// TIA Portal V21 export
FUNCTION "Cabinet_Management" : Void   // FC1, LAD
{ S7_Optimized_Access := 'TRUE' }
// stored: SetENOAutomatically false
   VAR_TEMP
      Phase_monitor_OK : Bool;
      Auxiliary_sevices_OK : Bool;
      "400V_protections_OK" : Bool;
      "400V_power_lines_activated" : Bool;
      Aux_emergencies : Bool;
      Emergencies_OK : Bool;
      Aux_cabinet_OK : Bool;
      Cabinet_OK : Bool;
      Heater_OK : Bool;
      Insulation_Monitor_OK : Bool;
      Power_wrapping_machine_OK : Bool;
      Power_fast_doors_OK : Bool;
      Facility_fault : Bool;
      Summary_fault : Bool;
   END_VAR
   VAR_TEMP   // added for the SCL form of the ladder/FBD networks
      _w1 : Bool;
      _w2 : Bool;
   END_VAR
BEGIN

REGION Network 1: Cabinet power control
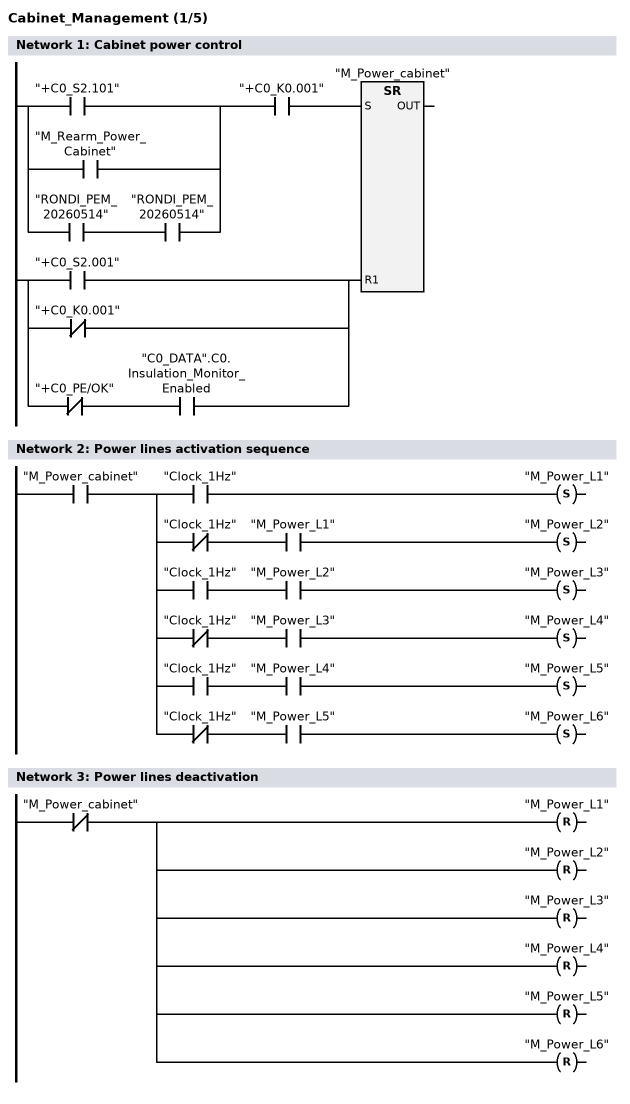
   RUNG wire#powerrail
      Contact( "+C0_S2.101" )
      wire#w1
      Contact( "+C0_K0.001" )
      S_SR(operand := "M_Power_cabinet", r1 := wire#w2)
   END_RUNG
   RUNG wire#powerrail
      Contact( "M_Rearm_Power_Cabinet" )
   END_RUNG wire#w1
   RUNG wire#powerrail
      Contact( "RONDI_PEM_20260514" )
      Contact( "RONDI_PEM_20260514" )
   END_RUNG wire#w1
   RUNG wire#powerrail
      Contact( "+C0_S2.001" )
   END_RUNG wire#w2
   RUNG wire#powerrail
      I_Contact( "+C0_K0.001" )
   END_RUNG wire#w2
   RUNG wire#powerrail
      I_Contact( "+C0_PE/OK" )
      Contact( "C0_DATA".C0.Insulation_Monitor_Enabled )
   END_RUNG wire#w2
   // the same network as SCL:
   IF ("+C0_S2.101" OR "M_Rearm_Power_Cabinet" OR ("RONDI_PEM_20260514" AND "RONDI_PEM_20260514")) AND "+C0_K0.001" THEN
       "M_Power_cabinet" := TRUE;   // SR flip-flop
   END_IF;
   IF "+C0_S2.001" OR NOT "+C0_K0.001" OR (NOT "+C0_PE/OK" AND "C0_DATA".C0.Insulation_Monitor_Enabled) THEN
       "M_Power_cabinet" := FALSE;
   END_IF;
END_REGION

REGION Network 2: Power lines activation sequence
   RUNG wire#powerrail
      Contact( "M_Power_cabinet" )
      wire#w1
      Contact( "Clock_1Hz" )
      S_Coil( "M_Power_L1" )
   END_RUNG
   RUNG wire#w1
      I_Contact( "Clock_1Hz" )
      Contact( "M_Power_L1" )
      S_Coil( "M_Power_L2" )
   END_RUNG
   RUNG wire#w1
      Contact( "Clock_1Hz" )
      Contact( "M_Power_L2" )
      S_Coil( "M_Power_L3" )
   END_RUNG
   RUNG wire#w1
      I_Contact( "Clock_1Hz" )
      Contact( "M_Power_L3" )
      S_Coil( "M_Power_L4" )
   END_RUNG
   RUNG wire#w1
      Contact( "Clock_1Hz" )
      Contact( "M_Power_L4" )
      S_Coil( "M_Power_L5" )
   END_RUNG
   RUNG wire#w1
      I_Contact( "Clock_1Hz" )
      Contact( "M_Power_L5" )
      S_Coil( "M_Power_L6" )
   END_RUNG
   // the same network as SCL:
   IF "M_Power_cabinet" AND "Clock_1Hz" THEN "M_Power_L1" := TRUE; END_IF;
   IF "M_Power_cabinet" AND NOT "Clock_1Hz" AND "M_Power_L1" THEN "M_Power_L2" := TRUE; END_IF;
   IF "M_Power_cabinet" AND "Clock_1Hz" AND "M_Power_L2" THEN "M_Power_L3" := TRUE; END_IF;
   IF "M_Power_cabinet" AND NOT "Clock_1Hz" AND "M_Power_L3" THEN "M_Power_L4" := TRUE; END_IF;
   IF "M_Power_cabinet" AND "Clock_1Hz" AND "M_Power_L4" THEN "M_Power_L5" := TRUE; END_IF;
   IF "M_Power_cabinet" AND NOT "Clock_1Hz" AND "M_Power_L5" THEN "M_Power_L6" := TRUE; END_IF;
END_REGION

REGION Network 3: Power lines deactivation
   RUNG wire#powerrail
      I_Contact( "M_Power_cabinet" )
      wire#w1
      R_Coil( "M_Power_L1" )
   END_RUNG
   RUNG wire#w1
      R_Coil( "M_Power_L2" )
   END_RUNG
   RUNG wire#w1
      R_Coil( "M_Power_L3" )
   END_RUNG
   RUNG wire#w1
      R_Coil( "M_Power_L4" )
   END_RUNG
   RUNG wire#w1
      R_Coil( "M_Power_L5" )
   END_RUNG
   RUNG wire#w1
      R_Coil( "M_Power_L6" )
   END_RUNG
   // the same network as SCL:
   IF NOT "M_Power_cabinet" THEN
       "M_Power_L1" := FALSE;
       "M_Power_L2" := FALSE;
       "M_Power_L3" := FALSE;
       "M_Power_L4" := FALSE;
       "M_Power_L5" := FALSE;
       "M_Power_L6" := FALSE;
   END_IF;
END_REGION

REGION Network 4: Power lines outputs
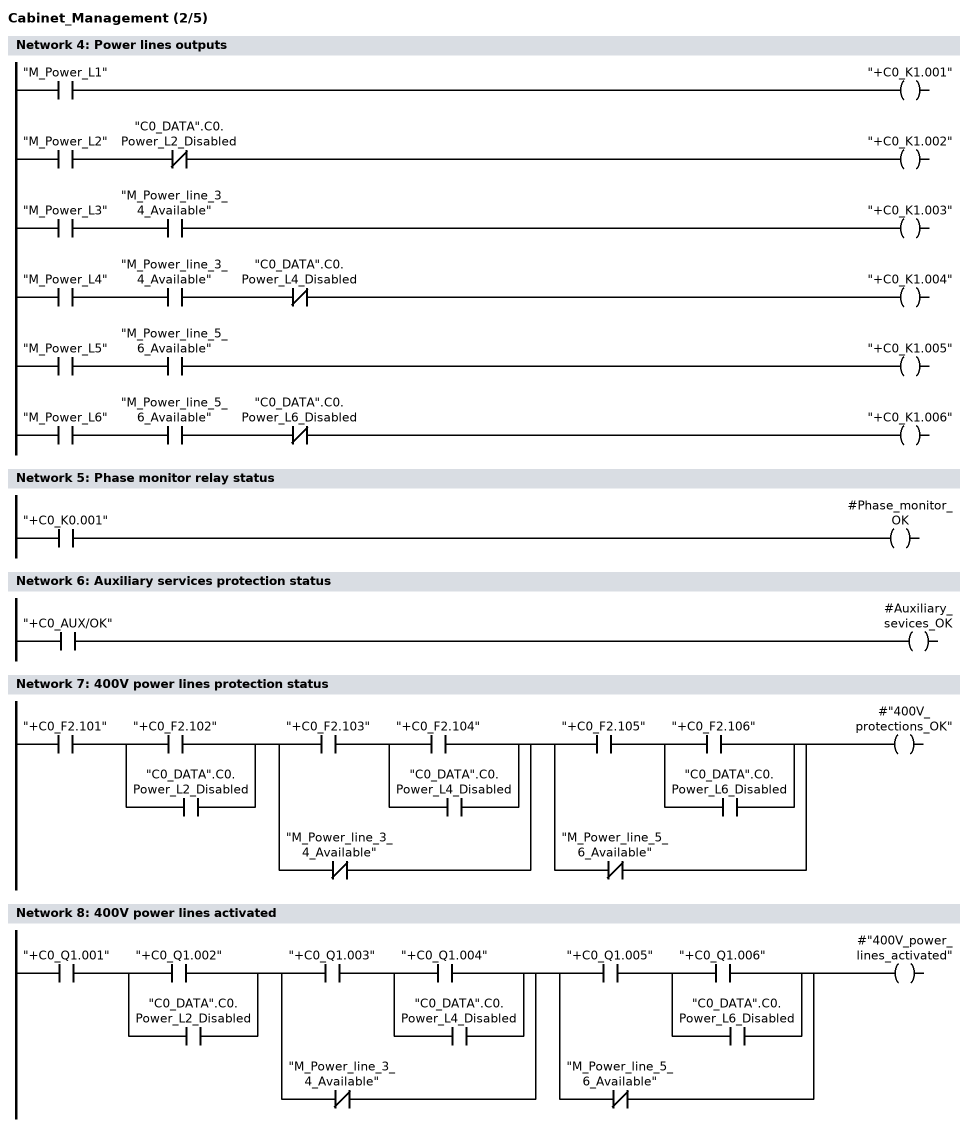
   RUNG wire#powerrail
      Contact( "M_Power_L1" )
      Coil( "+C0_K1.001" )
   END_RUNG
   RUNG wire#powerrail
      Contact( "M_Power_L2" )
      I_Contact( "C0_DATA".C0.Power_L2_Disabled )
      Coil( "+C0_K1.002" )
   END_RUNG
   RUNG wire#powerrail
      Contact( "M_Power_L3" )
      Contact( "M_Power_line_3_4_Available" )
      Coil( "+C0_K1.003" )
   END_RUNG
   RUNG wire#powerrail
      Contact( "M_Power_L4" )
      Contact( "M_Power_line_3_4_Available" )
      I_Contact( "C0_DATA".C0.Power_L4_Disabled )
      Coil( "+C0_K1.004" )
   END_RUNG
   RUNG wire#powerrail
      Contact( "M_Power_L5" )
      Contact( "M_Power_line_5_6_Available" )
      Coil( "+C0_K1.005" )
   END_RUNG
   RUNG wire#powerrail
      Contact( "M_Power_L6" )
      Contact( "M_Power_line_5_6_Available" )
      I_Contact( "C0_DATA".C0.Power_L6_Disabled )
      Coil( "+C0_K1.006" )
   END_RUNG
   // the same network as SCL:
   "+C0_K1.001" := "M_Power_L1";
   "+C0_K1.002" := "M_Power_L2" AND NOT "C0_DATA".C0.Power_L2_Disabled;
   "+C0_K1.003" := "M_Power_L3" AND "M_Power_line_3_4_Available";
   "+C0_K1.004" := "M_Power_L4" AND "M_Power_line_3_4_Available" AND NOT "C0_DATA".C0.Power_L4_Disabled;
   "+C0_K1.005" := "M_Power_L5" AND "M_Power_line_5_6_Available";
   "+C0_K1.006" := "M_Power_L6" AND "M_Power_line_5_6_Available" AND NOT "C0_DATA".C0.Power_L6_Disabled;
END_REGION

REGION Network 5: Phase monitor relay status
   RUNG wire#powerrail
      Contact( "+C0_K0.001" )
      Coil( #Phase_monitor_OK )
   END_RUNG
   // the same network as SCL:
   #Phase_monitor_OK := "+C0_K0.001";
END_REGION

REGION Network 6: Auxiliary services protection status
   RUNG wire#powerrail
      Contact( "+C0_AUX/OK" )
      Coil( #Auxiliary_sevices_OK )
   END_RUNG
   // the same network as SCL:
   #Auxiliary_sevices_OK := "+C0_AUX/OK";
END_REGION

REGION Network 7: 400V power lines protection status
   RUNG wire#powerrail
      Contact( "+C0_F2.101" )
      wire#w1
      Contact( "+C0_F2.102" )
      wire#w2
      Contact( "+C0_F2.103" )
      wire#w3
      Contact( "+C0_F2.104" )
      wire#w4
      Contact( "+C0_F2.105" )
      wire#w5
      Contact( "+C0_F2.106" )
      wire#w6
      Coil( #"400V_protections_OK" )
   END_RUNG
   RUNG wire#w1
      Contact( "C0_DATA".C0.Power_L2_Disabled )
   END_RUNG wire#w2
   RUNG wire#w3
      Contact( "C0_DATA".C0.Power_L4_Disabled )
   END_RUNG wire#w4
   RUNG wire#w2
      I_Contact( "M_Power_line_3_4_Available" )
   END_RUNG wire#w4
   RUNG wire#w5
      Contact( "C0_DATA".C0.Power_L6_Disabled )
   END_RUNG wire#w6
   RUNG wire#w4
      I_Contact( "M_Power_line_5_6_Available" )
   END_RUNG wire#w6
   // the same network as SCL:
   #"400V_protections_OK" := "+C0_F2.101" AND ("+C0_F2.102" OR "C0_DATA".C0.Power_L2_Disabled) AND (("+C0_F2.103" AND ("+C0_F2.104" OR "C0_DATA".C0.Power_L4_Disabled)) OR NOT "M_Power_line_3_4_Available") AND (("+C0_F2.105" AND ("+C0_F2.106" OR "C0_DATA".C0.Power_L6_Disabled)) OR NOT "M_Power_line_5_6_Available");
END_REGION

REGION Network 8: 400V power lines activated
   RUNG wire#powerrail
      Contact( "+C0_Q1.001" )
      wire#w1
      Contact( "+C0_Q1.002" )
      wire#w2
      Contact( "+C0_Q1.003" )
      wire#w3
      Contact( "+C0_Q1.004" )
      wire#w4
      Contact( "+C0_Q1.005" )
      wire#w5
      Contact( "+C0_Q1.006" )
      wire#w6
      Coil( #"400V_power_lines_activated" )
   END_RUNG
   RUNG wire#w1
      Contact( "C0_DATA".C0.Power_L2_Disabled )
   END_RUNG wire#w2
   RUNG wire#w3
      Contact( "C0_DATA".C0.Power_L4_Disabled )
   END_RUNG wire#w4
   RUNG wire#w2
      I_Contact( "M_Power_line_3_4_Available" )
   END_RUNG wire#w4
   RUNG wire#w5
      Contact( "C0_DATA".C0.Power_L6_Disabled )
   END_RUNG wire#w6
   RUNG wire#w4
      I_Contact( "M_Power_line_5_6_Available" )
   END_RUNG wire#w6
   // the same network as SCL:
   #"400V_power_lines_activated" := "+C0_Q1.001" AND ("+C0_Q1.002" OR "C0_DATA".C0.Power_L2_Disabled) AND (("+C0_Q1.003" AND ("+C0_Q1.004" OR "C0_DATA".C0.Power_L4_Disabled)) OR NOT "M_Power_line_3_4_Available") AND (("+C0_Q1.005" AND ("+C0_Q1.006" OR "C0_DATA".C0.Power_L6_Disabled)) OR NOT "M_Power_line_5_6_Available");
END_REGION

REGION Network 9: Emergency stops + Safety lines status
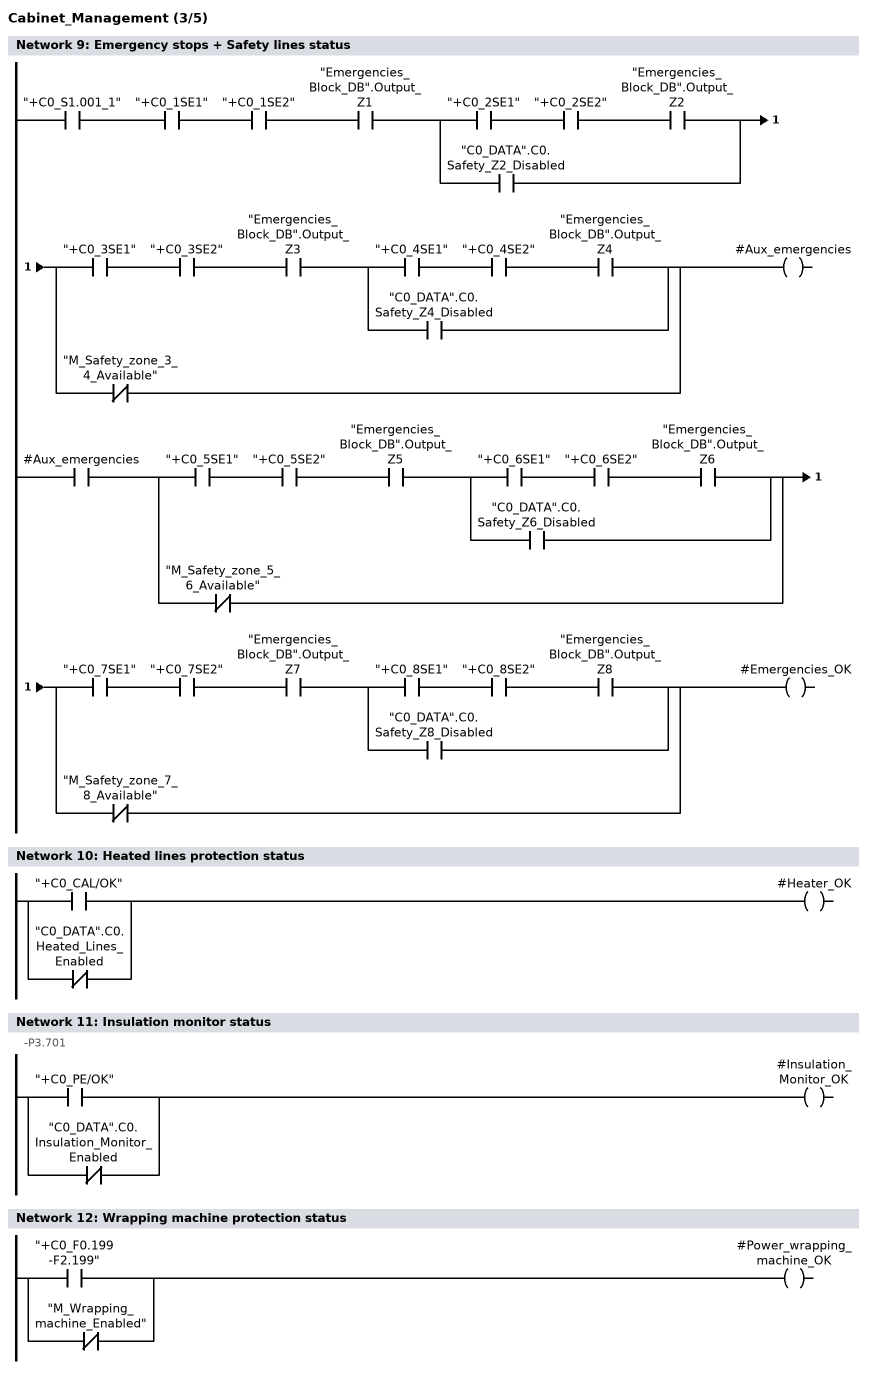
   RUNG wire#powerrail
      Contact( "+C0_S1.001_1" )
      Contact( "+C0_1SE1" )
      Contact( "+C0_1SE2" )
      Contact( "Emergencies_Block_DB".Output_Z1 )
      wire#w1
      Contact( "+C0_2SE1" )
      Contact( "+C0_2SE2" )
      Contact( "Emergencies_Block_DB".Output_Z2 )
      wire#w2
      Contact( "+C0_3SE1" )
      Contact( "+C0_3SE2" )
      Contact( "Emergencies_Block_DB".Output_Z3 )
      wire#w3
      Contact( "+C0_4SE1" )
      Contact( "+C0_4SE2" )
      Contact( "Emergencies_Block_DB".Output_Z4 )
      wire#w4
      Coil( #Aux_emergencies )
   END_RUNG
   RUNG wire#w1
      Contact( "C0_DATA".C0.Safety_Z2_Disabled )
   END_RUNG wire#w2
   RUNG wire#w3
      Contact( "C0_DATA".C0.Safety_Z4_Disabled )
   END_RUNG wire#w4
   RUNG wire#w2
      I_Contact( "M_Safety_zone_3_4_Available" )
   END_RUNG wire#w4
   RUNG wire#powerrail
      Contact( #Aux_emergencies )
      wire#w5
      Contact( "+C0_5SE1" )
      Contact( "+C0_5SE2" )
      Contact( "Emergencies_Block_DB".Output_Z5 )
      wire#w6
      Contact( "+C0_6SE1" )
      Contact( "+C0_6SE2" )
      Contact( "Emergencies_Block_DB".Output_Z6 )
      wire#w7
      Contact( "+C0_7SE1" )
      Contact( "+C0_7SE2" )
      Contact( "Emergencies_Block_DB".Output_Z7 )
      wire#w8
      Contact( "+C0_8SE1" )
      Contact( "+C0_8SE2" )
      Contact( "Emergencies_Block_DB".Output_Z8 )
      wire#w9
      Coil( #Emergencies_OK )
   END_RUNG
   RUNG wire#w6
      Contact( "C0_DATA".C0.Safety_Z6_Disabled )
   END_RUNG wire#w7
   RUNG wire#w5
      I_Contact( "M_Safety_zone_5_6_Available" )
   END_RUNG wire#w7
   RUNG wire#w8
      Contact( "C0_DATA".C0.Safety_Z8_Disabled )
   END_RUNG wire#w9
   RUNG wire#w7
      I_Contact( "M_Safety_zone_7_8_Available" )
   END_RUNG wire#w9
   // the same network as SCL:
   #Aux_emergencies := "+C0_S1.001_1" AND "+C0_1SE1" AND "+C0_1SE2" AND "Emergencies_Block_DB".Output_Z1 AND (("+C0_2SE1" AND "+C0_2SE2" AND "Emergencies_Block_DB".Output_Z2) OR "C0_DATA".C0.Safety_Z2_Disabled) AND (("+C0_3SE1" AND "+C0_3SE2" AND "Emergencies_Block_DB".Output_Z3 AND (("+C0_4SE1" AND "+C0_4SE2" AND "Emergencies_Block_DB".Output_Z4) OR "C0_DATA".C0.Safety_Z4_Disabled)) OR NOT "M_Safety_zone_3_4_Available");
   #Emergencies_OK := #Aux_emergencies AND (("+C0_5SE1" AND "+C0_5SE2" AND "Emergencies_Block_DB".Output_Z5 AND (("+C0_6SE1" AND "+C0_6SE2" AND "Emergencies_Block_DB".Output_Z6) OR "C0_DATA".C0.Safety_Z6_Disabled)) OR NOT "M_Safety_zone_5_6_Available") AND (("+C0_7SE1" AND "+C0_7SE2" AND "Emergencies_Block_DB".Output_Z7 AND (("+C0_8SE1" AND "+C0_8SE2" AND "Emergencies_Block_DB".Output_Z8) OR "C0_DATA".C0.Safety_Z8_Disabled)) OR NOT "M_Safety_zone_7_8_Available");
END_REGION

REGION Network 10: Heated lines protection status
   RUNG wire#powerrail
      Contact( "+C0_CAL/OK" )
      wire#w1
      Coil( #Heater_OK )
   END_RUNG
   RUNG wire#powerrail
      I_Contact( "C0_DATA".C0.Heated_Lines_Enabled )
   END_RUNG wire#w1
   // the same network as SCL:
   #Heater_OK := "+C0_CAL/OK" OR NOT "C0_DATA".C0.Heated_Lines_Enabled;
END_REGION

REGION Network 11: Insulation monitor status
   // -P3.701
   RUNG wire#powerrail
      Contact( "+C0_PE/OK" )
      wire#w1
      Coil( #Insulation_Monitor_OK )
   END_RUNG
   RUNG wire#powerrail
      I_Contact( "C0_DATA".C0.Insulation_Monitor_Enabled )
   END_RUNG wire#w1
   // the same network as SCL:
   #Insulation_Monitor_OK := "+C0_PE/OK" OR NOT "C0_DATA".C0.Insulation_Monitor_Enabled;
END_REGION

REGION Network 12: Wrapping machine protection status
   RUNG wire#powerrail
      Contact( "+C0_F0.199 -F2.199" )
      wire#w1
      Coil( #Power_wrapping_machine_OK )
   END_RUNG
   RUNG wire#powerrail
      I_Contact( "M_Wrapping_machine_Enabled" )
   END_RUNG wire#w1
   // the same network as SCL:
   #Power_wrapping_machine_OK := "+C0_F0.199 -F2.199" OR NOT "M_Wrapping_machine_Enabled";
END_REGION

REGION Network 13: Fast doors protection status
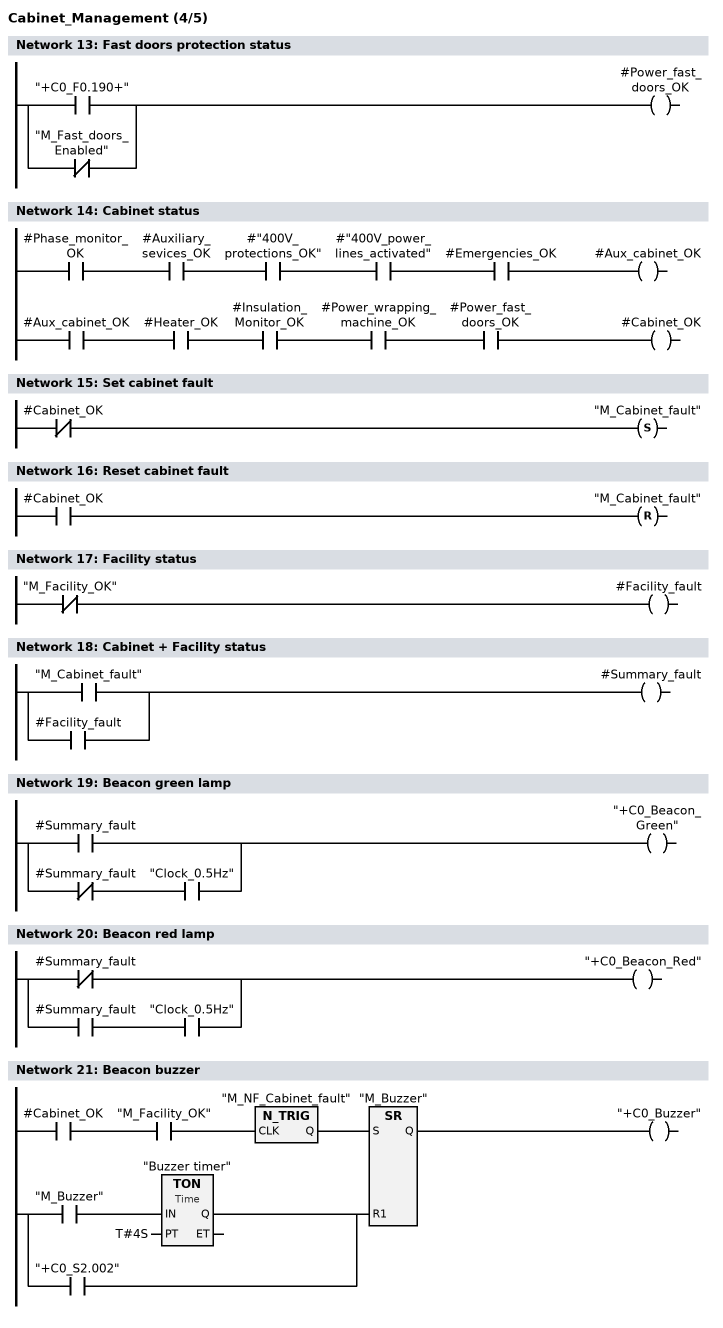
   RUNG wire#powerrail
      Contact( "+C0_F0.190+" )
      wire#w1
      Coil( #Power_fast_doors_OK )
   END_RUNG
   RUNG wire#powerrail
      I_Contact( "M_Fast_doors_Enabled" )
   END_RUNG wire#w1
   // the same network as SCL:
   #Power_fast_doors_OK := "+C0_F0.190+" OR NOT "M_Fast_doors_Enabled";
END_REGION

REGION Network 14: Cabinet status
   RUNG wire#powerrail
      Contact( #Phase_monitor_OK )
      Contact( #Auxiliary_sevices_OK )
      Contact( #"400V_protections_OK" )
      Contact( #"400V_power_lines_activated" )
      Contact( #Emergencies_OK )
      Coil( #Aux_cabinet_OK )
   END_RUNG
   RUNG wire#powerrail
      Contact( #Aux_cabinet_OK )
      Contact( #Heater_OK )
      Contact( #Insulation_Monitor_OK )
      Contact( #Power_wrapping_machine_OK )
      Contact( #Power_fast_doors_OK )
      Coil( #Cabinet_OK )
   END_RUNG
   // the same network as SCL:
   #Aux_cabinet_OK := #Phase_monitor_OK AND #Auxiliary_sevices_OK AND #"400V_protections_OK" AND #"400V_power_lines_activated" AND #Emergencies_OK;
   #Cabinet_OK := #Aux_cabinet_OK AND #Heater_OK AND #Insulation_Monitor_OK AND #Power_wrapping_machine_OK AND #Power_fast_doors_OK;
END_REGION

REGION Network 15: Set cabinet fault
   RUNG wire#powerrail
      I_Contact( #Cabinet_OK )
      S_Coil( "M_Cabinet_fault" )
   END_RUNG
   // the same network as SCL:
   IF NOT #Cabinet_OK THEN "M_Cabinet_fault" := TRUE; END_IF;
END_REGION

REGION Network 16: Reset cabinet fault
   RUNG wire#powerrail
      Contact( #Cabinet_OK )
      R_Coil( "M_Cabinet_fault" )
   END_RUNG
   // the same network as SCL:
   IF #Cabinet_OK THEN "M_Cabinet_fault" := FALSE; END_IF;
END_REGION

REGION Network 17: Facility status
   RUNG wire#powerrail
      I_Contact( "M_Facility_OK" )
      Coil( #Facility_fault )
   END_RUNG
   // the same network as SCL:
   #Facility_fault := NOT "M_Facility_OK";
END_REGION

REGION Network 18: Cabinet + Facility status
   RUNG wire#powerrail
      Contact( "M_Cabinet_fault" )
      wire#w1
      Coil( #Summary_fault )
   END_RUNG
   RUNG wire#powerrail
      Contact( #Facility_fault )
   END_RUNG wire#w1
   // the same network as SCL:
   #Summary_fault := "M_Cabinet_fault" OR #Facility_fault;
END_REGION

REGION Network 19: Beacon green lamp
   RUNG wire#powerrail
      Contact( #Summary_fault )
      wire#w1
      Coil( "+C0_Beacon_Green" )
   END_RUNG
   RUNG wire#powerrail
      I_Contact( #Summary_fault )
      Contact( "Clock_0.5Hz" )
   END_RUNG wire#w1
   // the same network as SCL:
   "+C0_Beacon_Green" := #Summary_fault OR (NOT #Summary_fault AND "Clock_0.5Hz");
END_REGION

REGION Network 20: Beacon red lamp
   RUNG wire#powerrail
      I_Contact( #Summary_fault )
      wire#w1
      Coil( "+C0_Beacon_Red" )
   END_RUNG
   RUNG wire#powerrail
      Contact( #Summary_fault )
      Contact( "Clock_0.5Hz" )
   END_RUNG wire#w1
   // the same network as SCL:
   "+C0_Beacon_Red" := NOT #Summary_fault OR (#Summary_fault AND "Clock_0.5Hz");
END_REGION

REGION Network 21: Beacon buzzer
   RUNG wire#powerrail
      Contact( #Cabinet_OK )
      Contact( "M_Facility_OK" )
      N_Trig( "M_NF_Cabinet_fault" )
      S_SR(operand := "M_Buzzer", r1 := wire#w1)
      Coil( "+C0_Buzzer" )
   END_RUNG
   RUNG wire#powerrail
      Contact( "M_Buzzer" )
      { S7_Templates := "time_type := Time" } "Buzzer timer".TON(pt := T#4S, et =>)
   END_RUNG wire#w1
   RUNG wire#powerrail
      Contact( "+C0_S2.002" )
   END_RUNG wire#w1
   // the same network as SCL:
   #_w1 := #Cabinet_OK AND "M_Facility_OK";
   #_w2 := NOT #_w1 AND "M_NF_Cabinet_fault";   // falling edge
   "M_NF_Cabinet_fault" := #_w1;
   "Buzzer timer".TON(IN := "M_Buzzer", PT := T#4S);
   IF #_w2 THEN
       "M_Buzzer" := TRUE;   // SR flip-flop
   END_IF;
   IF "Buzzer timer".Q OR "+C0_S2.002" THEN "M_Buzzer" := FALSE; END_IF;
   "+C0_Buzzer" := "M_Buzzer";
END_REGION

REGION Network 22: Cabinet power lines status indicator lamp
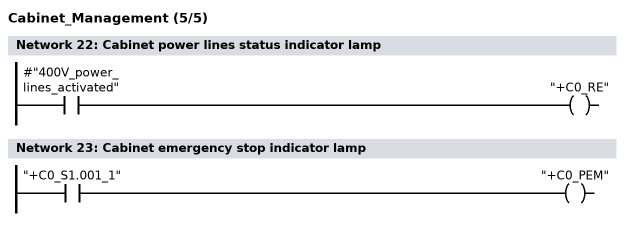
   RUNG wire#powerrail
      Contact( #"400V_power_lines_activated" )
      Coil( "+C0_RE" )
   END_RUNG
   // the same network as SCL:
   "+C0_RE" := #"400V_power_lines_activated";
END_REGION

REGION Network 23: Cabinet emergency stop indicator lamp
   RUNG wire#powerrail
      Contact( "+C0_S1.001_1" )
      Coil( "+C0_PEM" )
   END_RUNG
   // the same network as SCL:
   "+C0_PEM" := "+C0_S1.001_1";
END_REGION
END_FUNCTION
